FUNCTION_BLOCK SS1_ifb_Robot (* Basic FB with empty ECC *)
  (* Standard: 61499-2 *)
  (* Version 1.0, 2024-07-24, DEVIASH *)
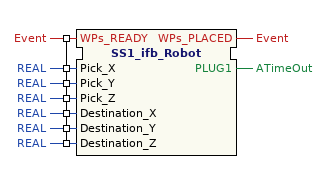
  EVENT_INPUT
    WPs_READY WITH Pick_X, Pick_Y, Pick_Z, Destination_X, Destination_Y, Destination_Z;
  END_EVENT
  EVENT_OUTPUT
    WPs_PLACED;
  END_EVENT
  VAR_INPUT
    Pick_X : REAL := 10.0;
    Pick_Y : REAL := 10.0;
    Pick_Z : REAL := 10.0;
    Destination_X : REAL := 10.0;
    Destination_Y : REAL := 10.0;
    Destination_Z : REAL := 10.0;
  END_VAR
  PLUGS
    PLUG1 : ATimeOut;
  END_PLUGS
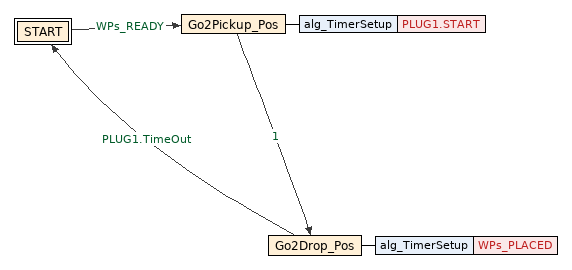
  EC_STATES
    START; (* Initial State *)
    Go2Pickup_Pos : alg_TimerSetup -> PLUG1.START;
    Go2Drop_Pos : alg_TimerSetup -> WPs_PLACED;
  END_STATES
  EC_TRANSITIONS
    START TO Go2Pickup_Pos := WPs_READY;
    Go2Pickup_Pos TO Go2Drop_Pos := 1;
    Go2Drop_Pos TO START := PLUG1.TimeOut;
  END_TRANSITIONS
  ALGORITHM alg_TimerSetup IN ST:
PLUG1.DT = T#5s;
  END_ALGORITHM
END_FUNCTION_BLOCK
